# EPICS substitutions: test/iocTest/TestApp/Db/test_mbbi.substitutions
file test_mbbi.template {
pattern
	{ DEV, INP_FIELD }

	{ "X", "@U0,S4,X1"}
	{ "Y", "@U0,S3,Y1"}
#	{ "A", "@U0,S3,A1"}
	{ "r", "@CPU2,R518"}
	{ "W", "@W10001"}
	{ "L", "@L00001"}
	{ "M", "@U0,S3,M1"}
	{ "E", "@E00265"}
	{ "R", "@R00528"}
}
